TYPE E_TMCM_SwitchConfig :
(
	Activated := 0, 
	Deactivated := 1,
	Inverted := 2
);
END_TYPE

(* stored: Version 1.1.0.1, ProductVersion 3.1.4024.11
   DUT E_TMCM_SwitchConfig: Id {7044eb9f-e638-45ea-a49f-50c1300d2fbd} *)
